	// Assert
	TestSuite.Test(__POUNAME()).AssertEqual(TEST_BOOL_TRUE, Success);
	TEST_DINT := 0;  // Buffer empty
	TestSuite.Test(__POUNAME()).AssertEqual(TEST_DINT, fbAnyBuffer.Metadata.elementCount);
END_IF
END_METHOD

// Element is removed but not copied when popDiscard=TRUE
METHOD PopDiscardTrue
VAR
	discardBuffer : BYTE;  // Can be any type when popDiscard=TRUE
END_VAR
IF TestSuite.Test(__POUNAME()).ExecuteTest() THEN
	// Arrange
	fbAnyBuffer.Clear();
	RawBuffer[TEST_LL+0] := 100;
	RawBuffer[TEST_LL+1] := 200;
	RawBuffer[TEST_LL+2] := 300;
	fbAnyBuffer.Metadata.elementCount := 3;
	discardBuffer := 0;

	// Act - Pop with discard=TRUE
	Success := fbAnyBuffer.PopRight(element := discardBuffer, popDiscard := TRUE);

	// Assert - Success but discardBuffer unchanged (no copy occurred)
	TestSuite.Test(__POUNAME()).AssertEqual(TEST_BOOL_TRUE, Success);
	TEST_DINT := 2;
	TestSuite.Test(__POUNAME()).AssertEqual(TEST_DINT, fbAnyBuffer.Metadata.elementCount);
	// Buffer should remain unchanged except last element cleared: [100, 200, 0]
	TEST_DINT := 100;
	TestSuite.Test(__POUNAME()).AssertEqual(TEST_DINT, RawBuffer[TEST_LL+0]);
	TEST_DINT := 200;
	TestSuite.Test(__POUNAME()).AssertEqual(TEST_DINT, RawBuffer[TEST_LL+1]);
	TEST_DINT := 0;
	TestSuite.Test(__POUNAME()).AssertEqual(TEST_DINT, RawBuffer[TEST_LL+2]);
END_IF
END_METHOD

// ElementCount decreases when popDiscard=TRUE
METHOD PopDiscardTrueDecrementsCount
VAR
	discardBuffer : DINT;
END_VAR
IF TestSuite.Test(__POUNAME()).ExecuteTest() THEN
	// Arrange
	fbAnyBuffer.Clear();
	RawBuffer[TEST_LL+0] := 100;
	RawBuffer[TEST_LL+1] := 200;
	RawBuffer[TEST_LL+2] := 300;
	fbAnyBuffer.Metadata.elementCount := 3;
	TEST_DINT := 3;
	TestSuite.Test(__POUNAME()).AssertEqual(TEST_DINT, fbAnyBuffer.Metadata.elementCount);

	// Act - Pop with discard=TRUE
	Success := fbAnyBuffer.PopRight(element := discardBuffer, popDiscard := TRUE);

	// Assert - Count decremented
	TestSuite.Test(__POUNAME()).AssertEqual(TEST_BOOL_TRUE, Success);
	TEST_DINT := 2;
	TestSuite.Test(__POUNAME()).AssertEqual(TEST_DINT, fbAnyBuffer.Metadata.elementCount);
END_IF
END_METHOD

// No element shifting occurs when popDiscard=TRUE (same as default)
METHOD PopDiscardTrueNoShift
VAR
	discardBuffer : DINT;
END_VAR
IF TestSuite.Test(__POUNAME()).ExecuteTest() THEN
	// Arrange
	fbAnyBuffer.Clear();
	RawBuffer[TEST_LL+0] := 10;
	RawBuffer[TEST_LL+1] := 20;
	RawBuffer[TEST_LL+2] := 30;
	RawBuffer[TEST_LL+3] := 40;
	fbAnyBuffer.Metadata.elementCount := 4;

	// Act - Pop with discard=TRUE
	Success := fbAnyBuffer.PopRight(element := discardBuffer, popDiscard := TRUE);

	// Assert - Elements stay in place (no shift)
	TestSuite.Test(__POUNAME()).AssertEqual(TEST_BOOL_TRUE, Success);
	TEST_DINT := 10;
	TestSuite.Test(__POUNAME()).AssertEqual(TEST_DINT, RawBuffer[TEST_LL+0]);
	TEST_DINT := 20;
	TestSuite.Test(__POUNAME()).AssertEqual(TEST_DINT, RawBuffer[TEST_LL+1]);
	TEST_DINT := 30;
	TestSuite.Test(__POUNAME()).AssertEqual(TEST_DINT, RawBuffer[TEST_LL+2]);
	TEST_DINT := 0;  // Last element cleared
	TestSuite.Test(__POUNAME()).AssertEqual(TEST_DINT, RawBuffer[TEST_LL+3]);
END_IF
END_METHOD

// No error when element size is wrong and popDiscard=TRUE
METHOD PopDiscardTrueSkipsTypeCheck
VAR
	wrongSizeBuffer : BYTE;  // Only 1 byte, but buffer expects DINT (4 bytes)
END_VAR
IF TestSuite.Test(__POUNAME()).ExecuteTest() THEN
	// Arrange
	fbAnyBuffer.Clear();
	RawBuffer[TEST_LL+0] := 100;
	RawBuffer[TEST_LL+1] := 200;
	fbAnyBuffer.Metadata.elementCount := 2;
	wrongSizeBuffer := 0;

	// Act - Pop with wrong type but popDiscard=TRUE (should succeed)
	Success := fbAnyBuffer.PopRight(element := wrongSizeBuffer, popDiscard := TRUE);

	// Assert - Should succeed despite type mismatch
	TestSuite.Test(__POUNAME()).AssertEqual(TEST_BOOL_TRUE, Success);
	TEST_DINT := 1;
	TestSuite.Test(__POUNAME()).AssertEqual(TEST_DINT, fbAnyBuffer.Metadata.elementCount);
END_IF
END_METHOD

// PopRight with wrong type succeeds when popDiscard=TRUE
METHOD PopDiscardWithWrongTypeSucceeds
VAR
	wrongTypeBuffer : INT;  // 2 bytes instead of 4
END_VAR
IF TestSuite.Test(__POUNAME()).ExecuteTest() THEN
	// Arrange
	fbAnyBuffer.Clear();
	RawBuffer[TEST_LL+0] := 999;
	RawBuffer[TEST_LL+1] := 888;
	fbAnyBuffer.Metadata.elementCount := 2;
	wrongTypeBuffer := 0;

	// Act - Pop with wrong type but popDiscard=TRUE
	Success := fbAnyBuffer.PopRight(element := wrongTypeBuffer, popDiscard := TRUE);

	// Assert - Should succeed
	TestSuite.Test(__POUNAME()).AssertEqual(TEST_BOOL_TRUE, Success);
	TEST_DINT := 1;
	TestSuite.Test(__POUNAME()).AssertEqual(TEST_DINT, fbAnyBuffer.Metadata.elementCount);
	// First element unchanged, last element cleared
	TEST_DINT := 999;
	TestSuite.Test(__POUNAME()).AssertEqual(TEST_DINT, RawBuffer[TEST_LL+0]);
	TEST_DINT := 0;
	TestSuite.Test(__POUNAME()).AssertEqual(TEST_DINT, RawBuffer[TEST_LL+1]);
END_IF
END_METHOD

// PopRight on empty buffer returns FALSE and does not modify buffer
METHOD PopFromEmptyBuffer
IF TestSuite.Test(__POUNAME()).ExecuteTest() THEN
	// Arrange - Clear buffer (elementCount = 0)
	fbAnyBuffer.Clear();
	ReturnedElement := 999;  // Set to non-zero to verify it is NOT overwritten

	// Act - Pop from empty buffer
	Success := fbAnyBuffer.PopRight(element := ReturnedElement);

	// Assert - Should fail because buffer is empty
	TestSuite.Test(__POUNAME()).AssertEqual(TEST_BOOL_FALSE, Success);

	// Element should remain unchanged (999) since pop failed
	TEST_DINT := 999;
	TestSuite.Test(__POUNAME()).AssertEqual(TEST_DINT, ReturnedElement);

	// All buffer positions should remain 0
	TEST_DINT := 0;
	TestSuite.Test(__POUNAME()).AssertEqual(TEST_DINT, RawBuffer[TEST_LL+0]);
	TestSuite.Test(__POUNAME()).AssertEqual(TEST_DINT, RawBuffer[TEST_LL+1]);
	TestSuite.Test(__POUNAME()).AssertEqual(TEST_DINT, RawBuffer[TEST_LL+2]);
	TestSuite.Test(__POUNAME()).AssertEqual(TEST_DINT, RawBuffer[TEST_LL+3]);
	TestSuite.Test(__POUNAME()).AssertEqual(TEST_DINT, RawBuffer[TEST_LL+4]);
END_IF
END_METHOD

// PopRight when buffer contains exactly one element
METHOD PopSingleElement
IF TestSuite.Test(__POUNAME()).ExecuteTest() THEN
	// Arrange - Only first element has data
	fbAnyBuffer.Clear();
	RawBuffer[TEST_LL+0] := 42;
	fbAnyBuffer.Metadata.elementCount := 1;
	ReturnedElement := 0;

	// Act
	Success := fbAnyBuffer.PopRight(element := ReturnedElement);

	// Assert - Should retrieve the single element
	TestSuite.Test(__POUNAME()).AssertEqual(TEST_BOOL_TRUE, Success);
	TEST_DINT := 42;
	TestSuite.Test(__POUNAME()).AssertEqual(TEST_DINT, ReturnedElement);

	// Buffer should now be completely empty
	TEST_DINT := 0;
	TestSuite.Test(__POUNAME()).AssertEqual(TEST_DINT, fbAnyBuffer.Metadata.elementCount);
	TestSuite.Test(__POUNAME()).AssertEqual(TEST_DINT, RawBuffer[TEST_LL+0]);
	TestSuite.Test(__POUNAME()).AssertEqual(TEST_DINT, RawBuffer[TEST_LL+1]);
	TestSuite.Test(__POUNAME()).AssertEqual(TEST_DINT, RawBuffer[TEST_LL+2]);
	TestSuite.Test(__POUNAME()).AssertEqual(TEST_DINT, RawBuffer[TEST_LL+3]);
	TestSuite.Test(__POUNAME()).AssertEqual(TEST_DINT, RawBuffer[TEST_LL+4]);
END_IF
END_METHOD

// PopRight can pop all elements until buffer is empty
METHOD PopUntilEmpty
VAR
	i : INT;
	ReturnedElement : DINT;
	testElement : DINT;
END_VAR
IF TestSuite.Test(__POUNAME()).ExecuteTest() THEN
	// Arrange - Fill buffer completely
	fbAnyBuffer.Clear();
	FOR i := 1 TO 5 DO
		testElement := TO_DINT(i * 100);
		fbAnyBuffer.PushRight(element := testElement);
	END_FOR

	// Act - Pop all elements
	FOR i := 5 TO 1 BY -1 DO
		Success := fbAnyBuffer.PopRight(element := ReturnedElement);
		TestSuite.Test(__POUNAME()).AssertEqual(TEST_BOOL_TRUE, Success);
		TEST_DINT := TO_DINT(i * 100);
		TestSuite.Test(__POUNAME()).AssertEqual(TEST_DINT, ReturnedElement);
	END_FOR

	// Assert - Buffer should be completely empty
	TEST_DINT := 0;
	TestSuite.Test(__POUNAME()).AssertEqual(TEST_DINT, fbAnyBuffer.Metadata.elementCount);

	// Try to pop from empty buffer
	Success := fbAnyBuffer.PopRight(element := ReturnedElement);
	TestSuite.Test(__POUNAME()).AssertEqual(TEST_BOOL_FALSE, Success);
END_IF
END_METHOD

// PopRight retrieves the last element from the buffer
METHOD RetrievesLastElement
IF TestSuite.Test(__POUNAME()).ExecuteTest() THEN
	// Arrange
	fbAnyBuffer.Clear();
	RawBuffer[TEST_LL+0] := 100;
	RawBuffer[TEST_LL+1] := 200;
	RawBuffer[TEST_LL+2] := 300;
	RawBuffer[TEST_LL+3] := 400;
	RawBuffer[TEST_LL+4] := 500;
	fbAnyBuffer.Metadata.elementCount := 5;
	ReturnedElement := 0;

	// Act
	Success := fbAnyBuffer.PopRight(element := ReturnedElement);

	// Assert
	TestSuite.Test(__POUNAME()).AssertEqual(TEST_BOOL_TRUE, Success);
	TEST_DINT := 500;
	TestSuite.Test(__POUNAME()).AssertEqual(TEST_DINT, ReturnedElement);
END_IF
END_METHOD

// PopRight returns TRUE when pop succeeds
METHOD ReturnsTrueOnSuccess
IF TestSuite.Test(__POUNAME()).ExecuteTest() THEN
	// Arrange
	fbAnyBuffer.Clear();
	RawBuffer[TEST_LL+0] := 100;
	fbAnyBuffer.Metadata.elementCount := 1;

	// Act
	Success := fbAnyBuffer.PopRight(element := ReturnedElement);

	// Assert
	TestSuite.Test(__POUNAME()).AssertEqual(TEST_BOOL_TRUE, Success);
END_IF
END_METHOD

// PopRight returns FALSE when element size doesn't match buffer element size
METHOD WrongSize
IF TestSuite.Test(__POUNAME()).ExecuteTest() THEN
	// Arrange
	fbAnyBuffer.Clear();
	RawBuffer[TEST_LL+0] := 100;
	fbAnyBuffer.Metadata.elementCount := 1;
	WrongSizeElement := 0;

	// Act - Pass an INT (2 bytes) to a DINT buffer (4 bytes)
	Success := fbAnyBuffer.PopRight(element := WrongSizeElement);

	// Assert
	TestSuite.Test(__POUNAME()).AssertEqual(TEST_BOOL_FALSE, Success);
END_IF
END_METHOD

END_PROGRAM

// ---- UnitTests/AnyBuffer/TEST_AnyBuffer_PushLeft.TcPOU
PROGRAM TEST_AnyBuffer_PushLeft

PushToEmptyBuffer();
PushToNonEmptyBuffer();
IncrementsElementCount();
ShiftsExistingElements();
ReturnsTrueOnSuccess();
ReturnsFalseOnFullBuffer();
ReturnsFalseOnWrongSize();
PreservesExistingData();
PushMultipleElements();
PushToFullBufferMinus1();
PushWhenFullCapacity();
PushZeroSizedElement();
PushWithDifferentDataTypes();
ConsecutivePushAndPopLeft();
ConsecutivePushAndPopRight();
ElementOrderAfterMultiplePushes();
FillBufferCompletely();

// LIFO behavior with alternating AppendLeft and PopLeft calls
METHOD ConsecutivePushAndPopLeft
VAR
	poppedValue : DINT;
END_VAR
IF TestSuite.Test(__POUNAME()).ExecuteTest() THEN
	// Arrange
	fbAnyBuffer.Clear();

	// Act - Append then Pop (LIFO: Last In First Out)
	AppendedElement := DINT#100;
	fbAnyBuffer.PushLeft(element := AppendedElement);  // [100]
	AppendedElement := DINT#200;
	fbAnyBuffer.PushLeft(element := AppendedElement);  // [200, 100]
	AppendedElement := DINT#300;
	fbAnyBuffer.PushLeft(element := AppendedElement);  // [300, 200, 100]
	fbAnyBuffer.PopLeft(element := poppedValue);  // Pop 300

	// Assert - Should pop the last appended value (300)
	TEST_DINT := 300;
	TestSuite.Test(__POUNAME()).AssertEqual(TEST_DINT, poppedValue);

	// Buffer should now be [200, 100]
	TEST_DINT := 200;
	TestSuite.Test(__POUNAME()).AssertEqual(TEST_DINT, RawBuffer[TEST_LL+0]);
	TEST_DINT := 100;
	TestSuite.Test(__POUNAME()).AssertEqual(TEST_DINT, RawBuffer[TEST_LL+1]);
	TEST_DINT := 2;
	TestSuite.Test(__POUNAME()).AssertEqual(TEST_DINT, fbAnyBuffer.Metadata.elementCount);
END_IF
END_METHOD

// FIFO behavior with alternating AppendLeft and PopRight calls
METHOD ConsecutivePushAndPopRight
VAR
	poppedValue : DINT;
END_VAR
IF TestSuite.Test(__POUNAME()).ExecuteTest() THEN
	// Arrange
	fbAnyBuffer.Clear();

	// Act - Append Left and Pop Right (FIFO from right)
	AppendedElement := DINT#100;
	fbAnyBuffer.PushLeft(element := AppendedElement);  // [100]
	AppendedElement := DINT#200;
	fbAnyBuffer.PushLeft(element := AppendedElement);  // [200, 100]
	AppendedElement := DINT#300;
	fbAnyBuffer.PushLeft(element := AppendedElement);  // [300, 200, 100]
	fbAnyBuffer.PopRight(element := poppedValue);  // Pop 100 (first appended)

	// Assert - Should pop the first appended value (100)
	TEST_DINT := 100;
	TestSuite.Test(__POUNAME()).AssertEqual(TEST_DINT, poppedValue);

	// Buffer should now be [300, 200]
	TEST_DINT := 300;
	TestSuite.Test(__POUNAME()).AssertEqual(TEST_DINT, RawBuffer[TEST_LL+0]);
	TEST_DINT := 200;
	TestSuite.Test(__POUNAME()).AssertEqual(TEST_DINT, RawBuffer[TEST_LL+1]);
	TEST_DINT := 2;
	TestSuite.Test(__POUNAME()).AssertEqual(TEST_DINT, fbAnyBuffer.Metadata.elementCount);
END_IF
END_METHOD

// AppendLeft maintains correct element order after multiple appends
METHOD ElementOrderAfterMultiplePushes
IF TestSuite.Test(__POUNAME()).ExecuteTest() THEN
	// Arrange
	fbAnyBuffer.Clear();

	// Act - Append 5 different values
	AppendedElement := DINT#1;
	fbAnyBuffer.PushLeft(element := AppendedElement);    // [1]
	AppendedElement := DINT#2;
	fbAnyBuffer.PushLeft(element := AppendedElement);    // [2, 1]
	AppendedElement := DINT#3;
	fbAnyBuffer.PushLeft(element := AppendedElement);    // [3, 2, 1]
	AppendedElement := DINT#4;
	fbAnyBuffer.PushLeft(element := AppendedElement);    // [4, 3, 2, 1]
	AppendedElement := DINT#5;
	fbAnyBuffer.PushLeft(element := AppendedElement);    // [5, 4, 3, 2, 1]

	// Assert - Verify complete LIFO order
	TEST_DINT := 5;
	TestSuite.Test(__POUNAME()).AssertEqual(TEST_DINT, RawBuffer[TEST_LL+0]);
	TEST_DINT := 4;
	TestSuite.Test(__POUNAME()).AssertEqual(TEST_DINT, RawBuffer[TEST_LL+1]);
	TEST_DINT := 3;
	TestSuite.Test(__POUNAME()).AssertEqual(TEST_DINT, RawBuffer[TEST_LL+2]);
	TEST_DINT := 2;
	TestSuite.Test(__POUNAME()).AssertEqual(TEST_DINT, RawBuffer[TEST_LL+3]);
	TEST_DINT := 1;
	TestSuite.Test(__POUNAME()).AssertEqual(TEST_DINT, RawBuffer[TEST_LL+4]);
	TEST_DINT := 5;
	TestSuite.Test(__POUNAME()).AssertEqual(TEST_DINT, fbAnyBuffer.Metadata.elementCount);
END_IF
END_METHOD

// Filling buffer to full capacity works correctly
METHOD FillBufferCompletely
VAR
	i : INT;
END_VAR
IF TestSuite.Test(__POUNAME()).ExecuteTest() THEN
	// Arrange
	fbAnyBuffer.Clear();

	// Act - Fill buffer completely
	FOR i := 1 TO 5 DO
		AppendedElement := TO_DINT(i * 100);
		Success := fbAnyBuffer.PushLeft(element := AppendedElement);
		TestSuite.Test(__POUNAME()).AssertEqual(TEST_BOOL_TRUE, Success);
	END_FOR

	// Assert - All elements in correct positions (reverse order due to left append)
	TEST_DINT := 500;
	TestSuite.Test(__POUNAME()).AssertEqual(TEST_DINT, RawBuffer[TEST_LL+0]);
	TEST_DINT := 400;
	TestSuite.Test(__POUNAME()).AssertEqual(TEST_DINT, RawBuffer[TEST_LL+1]);
	TEST_DINT := 300;
	TestSuite.Test(__POUNAME()).AssertEqual(TEST_DINT, RawBuffer[TEST_LL+2]);
	TEST_DINT := 200;
	TestSuite.Test(__POUNAME()).AssertEqual(TEST_DINT, RawBuffer[TEST_LL+3]);
	TEST_DINT := 100;
	TestSuite.Test(__POUNAME()).AssertEqual(TEST_DINT, RawBuffer[TEST_LL+4]);
	TEST_DINT := 5;
	TestSuite.Test(__POUNAME()).AssertEqual(TEST_DINT, fbAnyBuffer.Metadata.elementCount);

	// Assert - Cannot append when full
	AppendedElement := DINT#600;
	Success := fbAnyBuffer.PushLeft(element := AppendedElement);
	TestSuite.Test(__POUNAME()).AssertEqual(TEST_BOOL_FALSE, Success);
END_IF
END_METHOD

// AppendLeft increases elementCount by 1 after append
METHOD IncrementsElementCount
IF TestSuite.Test(__POUNAME()).ExecuteTest() THEN
	// Arrange
	fbAnyBuffer.Clear();
	RawBuffer[TEST_LL+0] := 100;
	RawBuffer[TEST_LL+1] := 200;
	fbAnyBuffer.Metadata.elementCount := 2;
	AppendedElement := 300;

	// Act
	Success := fbAnyBuffer.PushLeft(element := AppendedElement);

	// Assert - elementCount should be incremented from 2 to 3
	TEST_DINT := 3;
	TestSuite.Test(__POUNAME()).AssertEqual(TEST_DINT, fbAnyBuffer.Metadata.elementCount);
END_IF
END_METHOD

// AppendLeft preserves existing element values after shift
METHOD PreservesExistingData
IF TestSuite.Test(__POUNAME()).ExecuteTest() THEN
	// Arrange
	fbAnyBuffer.Clear();
	RawBuffer[TEST_LL+0] := 111;
	RawBuffer[TEST_LL+1] := 222;
	RawBuffer[TEST_LL+2] := 333;
	fbAnyBuffer.Metadata.elementCount := 3;
	AppendedElement := 999;

	// Act
	Success := fbAnyBuffer.PushLeft(element := AppendedElement);

	// Assert - All original values preserved (just shifted)
	TEST_DINT := 999;
	TestSuite.Test(__POUNAME()).AssertEqual(TEST_DINT, RawBuffer[TEST_LL+0]);
	TEST_DINT := 111;
	TestSuite.Test(__POUNAME()).AssertEqual(TEST_DINT, RawBuffer[TEST_LL+1]);
	TEST_DINT := 222;
	TestSuite.Test(__POUNAME()).AssertEqual(TEST_DINT, RawBuffer[TEST_LL+2]);
	TEST_DINT := 333;
	TestSuite.Test(__POUNAME()).AssertEqual(TEST_DINT, RawBuffer[TEST_LL+3]);
END_IF
END_METHOD

// AppendLeft consecutive appends work correctly (LIFO order)
METHOD PushMultipleElements
IF TestSuite.Test(__POUNAME()).ExecuteTest() THEN
	// Arrange
	fbAnyBuffer.Clear();

	// Act - Append multiple elements to the left (stack behavior)
	AppendedElement := DINT#10;
	fbAnyBuffer.PushLeft(element := AppendedElement);
	AppendedElement := DINT#20;
	fbAnyBuffer.PushLeft(element := AppendedElement);
	AppendedElement := DINT#30;
	fbAnyBuffer.PushLeft(element := AppendedElement);

	// Assert - LIFO order: last appended (30) should be at position 0
	TEST_DINT := 30;
	TestSuite.Test(__POUNAME()).AssertEqual(TEST_DINT, RawBuffer[TEST_LL+0]);
	TEST_DINT := 20;
	TestSuite.Test(__POUNAME()).AssertEqual(TEST_DINT, RawBuffer[TEST_LL+1]);
	TEST_DINT := 10;
	TestSuite.Test(__POUNAME()).AssertEqual(TEST_DINT, RawBuffer[TEST_LL+2]);
	TEST_DINT := 3;
	TestSuite.Test(__POUNAME()).AssertEqual(TEST_DINT, fbAnyBuffer.Metadata.elementCount);
END_IF
END_METHOD

// AppendLeft inserts element at position 0 in empty buffer
METHOD PushToEmptyBuffer
IF TestSuite.Test(__POUNAME()).ExecuteTest() THEN
	// Arrange
	fbAnyBuffer.Clear();
	AppendedElement := 100;

	// Act
	Success := fbAnyBuffer.PushLeft(element := AppendedElement);

	// Assert
	TestSuite.Test(__POUNAME()).AssertEqual(TEST_BOOL_TRUE, Success);
	TEST_DINT := 100;
	TestSuite.Test(__POUNAME()).AssertEqual(TEST_DINT, RawBuffer[TEST_LL+0]);
	TEST_DINT := 1;
	TestSuite.Test(__POUNAME()).AssertEqual(TEST_DINT, fbAnyBuffer.Metadata.elementCount);
END_IF
END_METHOD

// AppendLeft succeeds when buffer has exactly 1 space remaining
METHOD PushToFullBufferMinus1
IF TestSuite.Test(__POUNAME()).ExecuteTest() THEN
	// Arrange - Fill buffer with 4 elements (capacity is 5)
	fbAnyBuffer.Clear();
	RawBuffer[TEST_LL+0] := 100;
	RawBuffer[TEST_LL+1] := 200;
	RawBuffer[TEST_LL+2] := 300;
	RawBuffer[TEST_LL+3] := 400;
	fbAnyBuffer.Metadata.elementCount := 4;
	AppendedElement := 50;

	// Act - Append to buffer with exactly 1 space left
	Success := fbAnyBuffer.PushLeft(element := AppendedElement);

	// Assert
	TestSuite.Test(__POUNAME()).AssertEqual(TEST_BOOL_TRUE, Success);
	TEST_DINT := 5;
	TestSuite.Test(__POUNAME()).AssertEqual(TEST_DINT, fbAnyBuffer.Metadata.elementCount);
	TEST_DINT := 50;
	TestSuite.Test(__POUNAME()).AssertEqual(TEST_DINT, RawBuffer[TEST_LL+0]);
END_IF
END_METHOD

// AppendLeft inserts element at position 0 and shifts existing elements right
METHOD PushToNonEmptyBuffer
IF TestSuite.Test(__POUNAME()).ExecuteTest() THEN
	// Arrange
	fbAnyBuffer.Clear();
	RawBuffer[TEST_LL+0] := 200;
	RawBuffer[TEST_LL+1] := 300;
	fbAnyBuffer.Metadata.capacity := 3;
	fbAnyBuffer.Metadata.elementCount := 2;
	AppendedElement := 100;

	// Act
	Success := fbAnyBuffer.PushLeft(element := AppendedElement);

	// Assert
	TestSuite.Test(__POUNAME()).AssertEqual(TEST_BOOL_TRUE, Success);
	TEST_DINT := 100;
	TestSuite.Test(__POUNAME()).AssertEqual(TEST_DINT, RawBuffer[TEST_LL+0]);
	TEST_DINT := 200;
	TestSuite.Test(__POUNAME()).AssertEqual(TEST_DINT, RawBuffer[TEST_LL+1]);
	TEST_DINT := 300;
	TestSuite.Test(__POUNAME()).AssertEqual(TEST_DINT, RawBuffer[TEST_LL+2]);
END_IF
END_METHOD

// AppendLeft fails when elementCount equals capacity
METHOD PushWhenFullCapacity
IF TestSuite.Test(__POUNAME()).ExecuteTest() THEN
	// Arrange - Set elementCount to capacity
	// Arrange - Fill buffer to capacity (5 elements)
	fbAnyBuffer.Clear();
	RawBuffer[TEST_LL+0] := 100;
	RawBuffer[TEST_LL+1] := 200;
	RawBuffer[TEST_LL+2] := 300;
	RawBuffer[TEST_LL+3] := 400;
	RawBuffer[TEST_LL+4] := 500;
	fbAnyBuffer.Metadata.elementCount := TEST_UL-TEST_LL+1;
	fbAnyBuffer.Metadata.capacity := 0;
	AppendedElement := 999;

	// Act
	Success := fbAnyBuffer.PushLeft(element := AppendedElement);

	// Assert
	TestSuite.Test(__POUNAME()).AssertEqual(TEST_BOOL_FALSE, Success);
	TEST_DINT := 5;
	TestSuite.Test(__POUNAME()).AssertEqual(TEST_DINT, fbAnyBuffer.Metadata.elementCount);
END_IF
END_METHOD

// AppendLeft works with various data types (DINT, REAL, struct)
METHOD PushWithDifferentDataTypes
VAR
	realBuffer : ARRAY[0..4] OF REAL;
	fbRealBuffer : AnyBuffer(pBuffer := realBuffer,
								bufferBoundLower := 0,
								bufferBoundUpper := 4,
								isBufferPersistent := FALSE);
	realValue : REAL := 3.14159;
	retrievedReal : REAL;
END_VAR
IF TestSuite.Test(__POUNAME()).ExecuteTest() THEN
	// Arrange
	fbRealBuffer.Clear();
	realValue := 3.14159;

	// Act - Append REAL type
	Success := fbRealBuffer.PushLeft(element := realValue);

	// Assert
	TestSuite.Test(__POUNAME()).AssertEqual(TEST_BOOL_TRUE, Success);
	TEST_REAL := 3.14159;
	TestSuite.Test(__POUNAME()).AssertEqual(TEST_REAL, realBuffer[0]);
END_IF
END_METHOD

// AppendLeft with zero-sized element
METHOD PushZeroSizedElement
VAR
	EmptyAny				: __SYSTEM.AnyType;
END_VAR
IF TestSuite.Test(__POUNAME()).ExecuteTest() THEN
	// Arrange
	fbAnyBuffer.Clear();

	// Initialize empty AnyType (size = 0)
	EmptyAny.pValue := 0;
	EmptyAny.diSize := 0;

	// Act - Call with zero-sized element
	Success := fbAnyBuffer.PushLeft(element := EmptyAny);

	// Assert - Should fail because element size doesn't match
	TestSuite.Test(__POUNAME()).AssertEqual(TEST_BOOL_FALSE, Success);
END_IF
END_METHOD

// AppendLeft returns FALSE when buffer is at capacity
METHOD ReturnsFalseOnFullBuffer
IF TestSuite.Test(__POUNAME()).ExecuteTest() THEN
	// Arrange - Fill buffer to capacity (5 elements)
	fbAnyBuffer.Clear();
	RawBuffer[TEST_LL+0] := 100;
	RawBuffer[TEST_LL+1] := 200;
	RawBuffer[TEST_LL+2] := 300;
	RawBuffer[TEST_LL+3] := 400;
	RawBuffer[TEST_LL+4] := 500;
	fbAnyBuffer.Metadata.elementCount := TEST_UL+1;
	fbAnyBuffer.Metadata.capacity := 0;
	AppendedElement := 600;

	// Act - Try to append to full buffer
	Success := fbAnyBuffer.PushLeft(element := AppendedElement);

	// Assert
	TestSuite.Test(__POUNAME()).AssertEqual(TEST_BOOL_FALSE, Success);
	// Verify buffer unchanged
	TEST_DINT := 100;
	TestSuite.Test(__POUNAME()).AssertEqual(TEST_DINT, RawBuffer[TEST_LL+0]);
END_IF
END_METHOD

// AppendLeft returns FALSE when element size doesn't match buffer element size
METHOD ReturnsFalseOnWrongSize
IF TestSuite.Test(__POUNAME()).ExecuteTest() THEN
	// Arrange
	fbAnyBuffer.Clear();
	WrongSizeElement := 100;  // INT is 2 bytes, buffer expects DINT (4 bytes)

	// Act - Pass an INT to a DINT buffer
	Success := fbAnyBuffer.PushLeft(element := WrongSizeElement);

	// Assert
	TestSuite.Test(__POUNAME()).AssertEqual(TEST_BOOL_FALSE, Success);
END_IF
END_METHOD

// AppendLeft returns TRUE when append succeeds
METHOD ReturnsTrueOnSuccess
IF TestSuite.Test(__POUNAME()).ExecuteTest() THEN
	// Arrange
	fbAnyBuffer.Clear();
	AppendedElement := 42;

	// Act
	Success := fbAnyBuffer.PushLeft(element := AppendedElement);

	// Assert
	TestSuite.Test(__POUNAME()).AssertEqual(TEST_BOOL_TRUE, Success);
END_IF
END_METHOD

// AppendLeft shifts all existing elements right by one position
METHOD ShiftsExistingElements
IF TestSuite.Test(__POUNAME()).ExecuteTest() THEN
	// Arrange
	fbAnyBuffer.Clear();
	RawBuffer[TEST_LL+0] := 100;
	RawBuffer[TEST_LL+1] := 200;
	RawBuffer[TEST_LL+2] := 300;
	fbAnyBuffer.Metadata.elementCount := 3;
	AppendedElement := 50;

	// Act
	Success := fbAnyBuffer.PushLeft(element := AppendedElement);

	// Assert - all elements shifted right
	TEST_DINT := 50;
	TestSuite.Test(__POUNAME()).AssertEqual(TEST_DINT, RawBuffer[TEST_LL+0]);
	TEST_DINT := 100;
	TestSuite.Test(__POUNAME()).AssertEqual(TEST_DINT, RawBuffer[TEST_LL+1]);
	TEST_DINT := 200;
	TestSuite.Test(__POUNAME()).AssertEqual(TEST_DINT, RawBuffer[TEST_LL+2]);
	TEST_DINT := 300;
	TestSuite.Test(__POUNAME()).AssertEqual(TEST_DINT, RawBuffer[TEST_LL+3]);
END_IF
END_METHOD

END_PROGRAM

// ---- UnitTests/AnyBuffer/TEST_AnyBuffer_PushRight.TcPOU
PROGRAM TEST_AnyBuffer_PushRight

PushToEmptyBuffer();
PushToNonEmptyBuffer();
IncrementsElementCount();
DoesNotShiftElements();
ReturnsTrueOnSuccess();
ReturnsFalseOnFullBuffer();
ReturnsFalseOnWrongSize();
PreservesExistingData();
PushMultipleElements();
PushToFullBufferMinus1();
PushWhenFullCapacity();
PushZeroSizedElement();
PushWithDifferentDataTypes();
ConsecutivePushAndPopLeft();
ConsecutivePushAndPopRight();
ElementOrderAfterMultiplePushes();
FillBufferCompletely();

// AppendRight and PopLeft demonstrate FIFO behavior
METHOD ConsecutivePushAndPopLeft
VAR
	ReturnedElement : DINT;
END_VAR
IF TestSuite.Test(__POUNAME()).ExecuteTest() THEN
	// Arrange
	fbAnyBuffer.Clear();

	// Act - Append then Pop (FIFO: First In First Out)
	testElement := DINT#100;
	fbAnyBuffer.PushRight(element := testElement);  // [100]
	testElement := DINT#200;
	fbAnyBuffer.PushRight(element := testElement);  // [100, 200]
	testElement := DINT#300;
	fbAnyBuffer.PushRight(element := testElement);  // [100, 200, 300]
	fbAnyBuffer.PopLeft(element := ReturnedElement);   // Pop 100

	// Assert - Should pop the first appended value (100)
	TEST_DINT := 100;
	TestSuite.Test(__POUNAME()).AssertEqual(TEST_DINT, ReturnedElement);

	// Buffer should now be [200, 300]
	TEST_DINT := 200;
	TestSuite.Test(__POUNAME()).AssertEqual(TEST_DINT, RawBuffer[TEST_LL+0]);
	TEST_DINT := 300;
	TestSuite.Test(__POUNAME()).AssertEqual(TEST_DINT, RawBuffer[TEST_LL+1]);
END_IF
END_METHOD

// AppendRight and PopRight demonstrate LIFO behavior
METHOD ConsecutivePushAndPopRight
VAR
	ReturnedElement : DINT;
END_VAR
IF TestSuite.Test(__POUNAME()).ExecuteTest() THEN
	// Arrange
	fbAnyBuffer.Clear();

	// Act - Append then Pop from right (LIFO: Last In First Out)
	testElement := DINT#100;
	fbAnyBuffer.PushRight(element := testElement);  // [100]
	testElement := DINT#200;
	fbAnyBuffer.PushRight(element := testElement);  // [100, 200]
	testElement := DINT#300;
	fbAnyBuffer.PushRight(element := testElement);  // [100, 200, 300]
	fbAnyBuffer.PopRight(element := ReturnedElement);  // Pop 300

	// Assert - Should pop the last appended value (300)
	TEST_DINT := 300;
	TestSuite.Test(__POUNAME()).AssertEqual(TEST_DINT, ReturnedElement);

	// Buffer should now be [100, 200]
	TEST_DINT := 100;
	TestSuite.Test(__POUNAME()).AssertEqual(TEST_DINT, RawBuffer[TEST_LL+0]);
	TEST_DINT := 200;
	TestSuite.Test(__POUNAME()).AssertEqual(TEST_DINT, RawBuffer[TEST_LL+1]);
END_IF
END_METHOD

// AppendRight does not move any existing elements
METHOD DoesNotShiftElements
IF TestSuite.Test(__POUNAME()).ExecuteTest() THEN
	// Arrange
	fbAnyBuffer.Clear();
	RawBuffer[TEST_LL+0] := 111;
	RawBuffer[TEST_LL+1] := 222;
	RawBuffer[TEST_LL+2] := 333;
	fbAnyBuffer.Metadata.elementCount := 3;
	AppendedElement := 444;

	// Act
	Success := fbAnyBuffer.PushRight(element := AppendedElement);

	// Assert - all existing elements remain at their original positions
	TEST_DINT := 111;
	TestSuite.Test(__POUNAME()).AssertEqual(TEST_DINT, RawBuffer[TEST_LL+0]);
	TEST_DINT := 222;
	TestSuite.Test(__POUNAME()).AssertEqual(TEST_DINT, RawBuffer[TEST_LL+1]);
	TEST_DINT := 333;
	TestSuite.Test(__POUNAME()).AssertEqual(TEST_DINT, RawBuffer[TEST_LL+2]);
	TEST_DINT := 444;
	TestSuite.Test(__POUNAME()).AssertEqual(TEST_DINT, RawBuffer[TEST_LL+3]);
END_IF
END_METHOD

// AppendRight maintains correct element order after multiple appends
METHOD ElementOrderAfterMultiplePushes
IF TestSuite.Test(__POUNAME()).ExecuteTest() THEN
	// Arrange
	fbAnyBuffer.Clear();

	// Act - Append 5 different values
	testElement := DINT#1;
	fbAnyBuffer.PushRight(element := testElement);    // [1]
	testElement := DINT#2;
	fbAnyBuffer.PushRight(element := testElement);    // [1, 2]
	testElement := DINT#3;
	fbAnyBuffer.PushRight(element := testElement);    // [1, 2, 3]
	testElement := DINT#4;
	fbAnyBuffer.PushRight(element := testElement);    // [1, 2, 3, 4]
	testElement := DINT#5;
	fbAnyBuffer.PushRight(element := testElement);    // [1, 2, 3, 4, 5]

	// Assert - Verify sequential order
	TEST_DINT := 1;
	TestSuite.Test(__POUNAME()).AssertEqual(TEST_DINT, RawBuffer[TEST_LL+0]);
	TEST_DINT := 2;
	TestSuite.Test(__POUNAME()).AssertEqual(TEST_DINT, RawBuffer[TEST_LL+1]);
	TEST_DINT := 3;
	TestSuite.Test(__POUNAME()).AssertEqual(TEST_DINT, RawBuffer[TEST_LL+2]);
	TEST_DINT := 4;
	TestSuite.Test(__POUNAME()).AssertEqual(TEST_DINT, RawBuffer[TEST_LL+3]);
	TEST_DINT := 5;
	TestSuite.Test(__POUNAME()).AssertEqual(TEST_DINT, RawBuffer[TEST_LL+4]);
	TEST_DINT := 5;
	TestSuite.Test(__POUNAME()).AssertEqual(TEST_DINT, fbAnyBuffer.Metadata.elementCount);
END_IF
END_METHOD

// AppendRight can fill buffer to full capacity correctly
METHOD FillBufferCompletely
VAR
	i : INT;
END_VAR
IF TestSuite.Test(__POUNAME()).ExecuteTest() THEN
	// Arrange
	fbAnyBuffer.Clear();

	// Act - Fill buffer completely
	FOR i := 1 TO 5 DO
		testElement := TO_DINT(i * 100);
		Success := fbAnyBuffer.PushRight(element := testElement);
		TestSuite.Test(__POUNAME()).AssertEqual(TEST_BOOL_TRUE, Success);
	END_FOR

	// Assert - All elements in correct positions
	TEST_DINT := 100;
	TestSuite.Test(__POUNAME()).AssertEqual(TEST_DINT, RawBuffer[TEST_LL+0]);
	TEST_DINT := 200;
	TestSuite.Test(__POUNAME()).AssertEqual(TEST_DINT, RawBuffer[TEST_LL+1]);
	TEST_DINT := 300;
	TestSuite.Test(__POUNAME()).AssertEqual(TEST_DINT, RawBuffer[TEST_LL+2]);
	TEST_DINT := 400;
	TestSuite.Test(__POUNAME()).AssertEqual(TEST_DINT, RawBuffer[TEST_LL+3]);
	TEST_DINT := 500;
	TestSuite.Test(__POUNAME()).AssertEqual(TEST_DINT, RawBuffer[TEST_LL+4]);
	TEST_DINT := 5;
	TestSuite.Test(__POUNAME()).AssertEqual(TEST_DINT, fbAnyBuffer.Metadata.elementCount);

	// Assert - Cannot append when full
	testElement := DINT#600;
	Success := fbAnyBuffer.PushRight(element := testElement);
	TestSuite.Test(__POUNAME()).AssertEqual(TEST_BOOL_FALSE, Success);
END_IF
END_METHOD

// AppendRight increases elementCount by 1 after append
METHOD IncrementsElementCount
IF TestSuite.Test(__POUNAME()).ExecuteTest() THEN
	// Arrange
	fbAnyBuffer.Clear();
	RawBuffer[TEST_LL+0] := 100;
	RawBuffer[TEST_LL+1] := 200;
	fbAnyBuffer.Metadata.elementCount := 2;
	AppendedElement := 300;

	// Act
	Success := fbAnyBuffer.PushRight(element := AppendedElement);

	// Assert - elementCount should be incremented from 2 to 3
	TEST_DINT := 3;
	TestSuite.Test(__POUNAME()).AssertEqual(TEST_DINT, fbAnyBuffer.Metadata.elementCount);
END_IF
END_METHOD

// AppendRight preserves existing element values
METHOD PreservesExistingData
IF TestSuite.Test(__POUNAME()).ExecuteTest() THEN
	// Arrange
	fbAnyBuffer.Clear();
	RawBuffer[TEST_LL+0] := 111;
	RawBuffer[TEST_LL+1] := 222;
	RawBuffer[TEST_LL+2] := 333;
	fbAnyBuffer.Metadata.elementCount := 3;
	AppendedElement := 999;

	// Act
	Success := fbAnyBuffer.PushRight(element := AppendedElement);

	// Assert - All original values preserved (not shifted)
	TEST_DINT := 111;
	TestSuite.Test(__POUNAME()).AssertEqual(TEST_DINT, RawBuffer[TEST_LL+0]);
	TEST_DINT := 222;
	TestSuite.Test(__POUNAME()).AssertEqual(TEST_DINT, RawBuffer[TEST_LL+1]);
	TEST_DINT := 333;
	TestSuite.Test(__POUNAME()).AssertEqual(TEST_DINT, RawBuffer[TEST_LL+2]);
	TEST_DINT := 999;
	TestSuite.Test(__POUNAME()).AssertEqual(TEST_DINT, RawBuffer[TEST_LL+3]);
END_IF
END_METHOD

// AppendRight consecutive appends work correctly (FIFO order with PopLeft)
METHOD PushMultipleElements
IF TestSuite.Test(__POUNAME()).ExecuteTest() THEN
	// Arrange
	fbAnyBuffer.Clear();

	// Act - Append multiple elements to the right (queue behavior)
	testElement := DINT#10;
	fbAnyBuffer.PushRight(element := testElement);
	testElement := DINT#20;
	fbAnyBuffer.PushRight(element := testElement);
	testElement := DINT#30;
	fbAnyBuffer.PushRight(element := testElement);

	// Assert - Sequential order: elements appear in order appended
	TEST_DINT := 10;
	TestSuite.Test(__POUNAME()).AssertEqual(TEST_DINT, RawBuffer[TEST_LL+0]);
	TEST_DINT := 20;
	TestSuite.Test(__POUNAME()).AssertEqual(TEST_DINT, RawBuffer[TEST_LL+1]);
	TEST_DINT := 30;
	TestSuite.Test(__POUNAME()).AssertEqual(TEST_DINT, RawBuffer[TEST_LL+2]);
	TEST_DINT := 3;
	TestSuite.Test(__POUNAME()).AssertEqual(TEST_DINT, fbAnyBuffer.Metadata.elementCount);
END_IF
END_METHOD

// AppendRight inserts element at position 0 in empty buffer
METHOD PushToEmptyBuffer
IF TestSuite.Test(__POUNAME()).ExecuteTest() THEN
	// Arrange
	fbAnyBuffer.Clear();
	AppendedElement := 100;

	// Act
	Success := fbAnyBuffer.PushRight(element := AppendedElement);

	// Assert
	TestSuite.Test(__POUNAME()).AssertEqual(TEST_BOOL_TRUE, Success);
	TEST_DINT := 100;
	TestSuite.Test(__POUNAME()).AssertEqual(TEST_DINT, RawBuffer[TEST_LL+0]);
	TEST_DINT := 1;
	TestSuite.Test(__POUNAME()).AssertEqual(TEST_DINT, fbAnyBuffer.Metadata.elementCount);
END_IF
END_METHOD

// AppendRight succeeds when buffer has exactly 1 space remaining
METHOD PushToFullBufferMinus1
IF TestSuite.Test(__POUNAME()).ExecuteTest() THEN
	// Arrange - Fill buffer with 4 elements (capacity is 5)
	fbAnyBuffer.Clear();
	RawBuffer[TEST_LL+0] := 100;
	RawBuffer[TEST_LL+1] := 200;
	RawBuffer[TEST_LL+2] := 300;
	RawBuffer[TEST_LL+3] := 400;
	fbAnyBuffer.Metadata.elementCount := 4;
	AppendedElement := 500;

	// Act - Append to buffer with exactly 1 space left
	Success := fbAnyBuffer.PushRight(element := AppendedElement);

	// Assert
	TestSuite.Test(__POUNAME()).AssertEqual(TEST_BOOL_TRUE, Success);
	TEST_DINT := 5;
	TestSuite.Test(__POUNAME()).AssertEqual(TEST_DINT, fbAnyBuffer.Metadata.elementCount);
	TEST_DINT := 500;
	TestSuite.Test(__POUNAME()).AssertEqual(TEST_DINT, RawBuffer[TEST_LL+4]);
END_IF
END_METHOD

// AppendRight inserts element at position elementCount and no elements shift
METHOD PushToNonEmptyBuffer
IF TestSuite.Test(__POUNAME()).ExecuteTest() THEN
	// Arrange
	fbAnyBuffer.Clear();
	RawBuffer[TEST_LL+0] := 100;
	RawBuffer[TEST_LL+1] := 200;
	fbAnyBuffer.Metadata.capacity := 3;
	fbAnyBuffer.Metadata.elementCount := 2;
	AppendedElement := 300;

	// Act
	Success := fbAnyBuffer.PushRight(element := AppendedElement);

	// Assert
	TestSuite.Test(__POUNAME()).AssertEqual(TEST_BOOL_TRUE, Success);
	TEST_DINT := 100;
	TestSuite.Test(__POUNAME()).AssertEqual(TEST_DINT, RawBuffer[TEST_LL+0]);
	TEST_DINT := 200;
	TestSuite.Test(__POUNAME()).AssertEqual(TEST_DINT, RawBuffer[TEST_LL+1]);
	TEST_DINT := 300;
	TestSuite.Test(__POUNAME()).AssertEqual(TEST_DINT, RawBuffer[TEST_LL+2]);
END_IF
END_METHOD

// AppendRight fails when elementCount equals capacity
METHOD PushWhenFullCapacity
IF TestSuite.Test(__POUNAME()).ExecuteTest() THEN
	// Arrange - Fill buffer to capacity (5 elements)
	fbAnyBuffer.Clear();
	RawBuffer[TEST_LL+0] := 100;
	RawBuffer[TEST_LL+1] := 200;
	RawBuffer[TEST_LL+2] := 300;
	RawBuffer[TEST_LL+3] := 400;
	RawBuffer[TEST_LL+4] := 500;
	fbAnyBuffer.Metadata.elementCount := TEST_UL-TEST_LL+1;
	fbAnyBuffer.Metadata.capacity := 0;
	AppendedElement := 999;

	// Act
	Success := fbAnyBuffer.PushRight(element := AppendedElement);

	// Assert
	TestSuite.Test(__POUNAME()).AssertEqual(TEST_BOOL_FALSE, Success);
	TEST_DINT := 5;
	TestSuite.Test(__POUNAME()).AssertEqual(TEST_DINT, fbAnyBuffer.Metadata.elementCount);
END_IF
END_METHOD

// AppendRight works with various data types (DINT, REAL, struct)
METHOD PushWithDifferentDataTypes
VAR
	realBuffer : ARRAY[0..4] OF REAL;
	fbRealBuffer : AnyBuffer(pBuffer := realBuffer,
								bufferBoundLower := 0,
								bufferBoundUpper := 4,
								isBufferPersistent := FALSE);
	realValue : REAL := 3.14159;
	retrievedReal : REAL;
END_VAR
IF TestSuite.Test(__POUNAME()).ExecuteTest() THEN
	// Arrange
	fbRealBuffer.Clear();
	realValue := 3.14159;

	// Act - Append REAL type
	Success := fbRealBuffer.PushRight(element := realValue);

	// Assert
	TestSuite.Test(__POUNAME()).AssertEqual(TEST_BOOL_TRUE, Success);
	TEST_REAL := 3.14159;
	TestSuite.Test(__POUNAME()).AssertEqual(TEST_REAL, realBuffer[0]);
END_IF
END_METHOD

// AppendRight with zero-sized element
METHOD PushZeroSizedElement
VAR
	EmptyAny				: __SYSTEM.AnyType;
END_VAR
IF TestSuite.Test(__POUNAME()).ExecuteTest() THEN
	// Arrange
	fbAnyBuffer.Clear();

	// Initialize empty AnyType (size = 0)
	EmptyAny.pValue := 0;
	EmptyAny.diSize := 0;

	// Act - Call with zero-sized element
	Success := fbAnyBuffer.PushRight(element := EmptyAny);

	// Assert - Should fail because element size doesn't match
	TestSuite.Test(__POUNAME()).AssertEqual(TEST_BOOL_FALSE, Success);
END_IF
END_METHOD

// AppendRight returns FALSE when buffer is at capacity
METHOD ReturnsFalseOnFullBuffer
IF TestSuite.Test(__POUNAME()).ExecuteTest() THEN
	// Arrange - Fill buffer to capacity (5 elements)
	fbAnyBuffer.Clear();
	RawBuffer[TEST_LL+0] := 100;
	RawBuffer[TEST_LL+1] := 200;
	RawBuffer[TEST_LL+2] := 300;
	RawBuffer[TEST_LL+3] := 400;
	RawBuffer[TEST_LL+4] := 500;
	fbAnyBuffer.Metadata.elementCount := TEST_UL+1;
	fbAnyBuffer.Metadata.capacity := 0;
	AppendedElement := 600;

	// Act - Try to append to full buffer
	Success := fbAnyBuffer.PushRight(element := AppendedElement);

	// Assert
	TestSuite.Test(__POUNAME()).AssertEqual(TEST_BOOL_FALSE, Success);
	// Verify buffer unchanged
	TEST_DINT := 100;
	TestSuite.Test(__POUNAME()).AssertEqual(TEST_DINT, RawBuffer[TEST_LL+0]);
END_IF
END_METHOD

// AppendRight returns FALSE when element size doesn't match buffer element size
METHOD ReturnsFalseOnWrongSize
IF TestSuite.Test(__POUNAME()).ExecuteTest() THEN
	// Arrange
	fbAnyBuffer.Clear();
	WrongSizeElement := 100;  // INT is 2 bytes, buffer expects DINT (4 bytes)

	// Act - Pass an INT to a DINT buffer
	Success := fbAnyBuffer.PushRight(element := WrongSizeElement);

	// Assert
	TestSuite.Test(__POUNAME()).AssertEqual(TEST_BOOL_FALSE, Success);
END_IF
END_METHOD

// AppendRight returns TRUE when append succeeds
METHOD ReturnsTrueOnSuccess
IF TestSuite.Test(__POUNAME()).ExecuteTest() THEN
	// Arrange
	fbAnyBuffer.Clear();
	AppendedElement := 42;

	// Act
	Success := fbAnyBuffer.PushRight(element := AppendedElement);

	// Assert
	TestSuite.Test(__POUNAME()).AssertEqual(TEST_BOOL_TRUE, Success);
END_IF
END_METHOD

END_PROGRAM

// ---- UnitTests/AnyBuffer/TEST_AnyBuffer_ReplaceAtIndex.TcPOU
PROGRAM TEST_AnyBuffer_ReplaceAtIndex
VAR
	// Loop counter
	i						: DINT;
END_VAR

ReplaceAtBeginning();
ReplaceInMiddle();
ReplaceAtEnd();
ReturnsTrueOnSuccess();
ReturnsFalseOnNegativeIndex();
ReturnsFalseOnIndexAtCapacity();
ReturnsFalseOnIndexAboveCapacity();
WrongElementSize();
BufferUnchangedExceptIndex();
MetadataUnchanged();
MultipleReplacements();
ReplaceAllCapacityPositions();
ReplaceWithDifferentValues();
ReplaceSameIndexMultipleTimes();
ReplaceEmptyPosition();
ReplaceWhenBufferEmpty();

// All other elements remain unchanged after replace
METHOD BufferUnchangedExceptIndex
IF TestSuite.Test(__POUNAME()).ExecuteTest() THEN
	// Arrange - [100, 200, 300, 400, 500]
	fbAnyBuffer.Clear();
	FOR i := 1 TO 5 DO
		testElement := i * 100;
		fbAnyBuffer.PushRight(element := testElement);
	END_FOR

	// Act - Replace middle element (index 2)
	testElement := DINT#999;
	Success := fbAnyBuffer.ReplaceAtIndex(index := TEST_LL+2, element := testElement);

	// Assert - Only index 2 should be changed
	TestSuite.Test(__POUNAME()).AssertEqual(TEST_BOOL_TRUE, Success);
	TEST_DINT := 100;
	TestSuite.Test(__POUNAME()).AssertEqual(TEST_DINT, RawBuffer[TEST_LL+0]);
	TEST_DINT := 200;
	TestSuite.Test(__POUNAME()).AssertEqual(TEST_DINT, RawBuffer[TEST_LL+1]);
	TEST_DINT := 999;
	TestSuite.Test(__POUNAME()).AssertEqual(TEST_DINT, RawBuffer[TEST_LL+2]);
	TEST_DINT := 400;
	TestSuite.Test(__POUNAME()).AssertEqual(TEST_DINT, RawBuffer[TEST_LL+3]);
	TEST_DINT := 500;
	TestSuite.Test(__POUNAME()).AssertEqual(TEST_DINT, RawBuffer[TEST_LL+4]);
END_IF
END_METHOD

// ElementCount and all metadata remain unchanged after replace
METHOD MetadataUnchanged
IF TestSuite.Test(__POUNAME()).ExecuteTest() THEN
	// Arrange
	fbAnyBuffer.Clear();
	FOR i := 1 TO TEST_UL-TEST_LL+1 DO
		testElement := i * 100;
		fbAnyBuffer.PushRight(element := testElement);
	END_FOR
	TEST_DINT := 5;
	TestSuite.Test(__POUNAME()).AssertEqual(TEST_DINT, fbAnyBuffer.Metadata.elementCount);
	// Verify capacity was updated by PushRight
	TEST_DINT := 0;
	TestSuite.Test(__POUNAME()).AssertEqual(TEST_DINT, fbAnyBuffer.Metadata.capacity);

	// Act - Replace several elements
	testElement := DINT#111;
	Success := fbAnyBuffer.ReplaceAtIndex(index := TEST_LL, element := testElement);
	TestSuite.Test(__POUNAME()).AssertEqual(TEST_BOOL_TRUE, Success);

	testElement := DINT#333;
	Success := fbAnyBuffer.ReplaceAtIndex(index := TEST_LL+2, element := testElement);
	TestSuite.Test(__POUNAME()).AssertEqual(TEST_BOOL_TRUE, Success);

	testElement := DINT#555;
	Success := fbAnyBuffer.ReplaceAtIndex(index := TEST_LL+4, element := testElement);
	TestSuite.Test(__POUNAME()).AssertEqual(TEST_BOOL_TRUE, Success);

	// Assert - All metadata should be unchanged
	TEST_DINT := 5;
	TestSuite.Test(__POUNAME()).AssertEqual(TEST_DINT, fbAnyBuffer.Metadata.elementCount);
	TEST_DINT := 0;
	TestSuite.Test(__POUNAME()).AssertEqual(TEST_DINT, fbAnyBuffer.Metadata.capacity);
END_IF
END_METHOD

// Sequential replacements at different indices work correctly
METHOD MultipleReplacements
IF TestSuite.Test(__POUNAME()).ExecuteTest() THEN
	// Arrange
	fbAnyBuffer.Clear();
	FOR i := 1 TO TEST_UL-TEST_LL+1 DO
		testElement := i * 100;
		fbAnyBuffer.PushRight(element := testElement);
	END_FOR

	// Act - Replace multiple positions
	testElement := DINT#111;
	Success := fbAnyBuffer.ReplaceAtIndex(index := TEST_LL, element := testElement);
	TestSuite.Test(__POUNAME()).AssertEqual(TEST_BOOL_TRUE, Success);

	testElement := DINT#222;
	Success := fbAnyBuffer.ReplaceAtIndex(index := TEST_LL+1, element := testElement);
	TestSuite.Test(__POUNAME()).AssertEqual(TEST_BOOL_TRUE, Success);

	testElement := DINT#555;
	Success := fbAnyBuffer.ReplaceAtIndex(index := TEST_LL+4, element := testElement);
	TestSuite.Test(__POUNAME()).AssertEqual(TEST_BOOL_TRUE, Success);

	// Assert - All replacements should be successful
	TEST_DINT := 111;
	TestSuite.Test(__POUNAME()).AssertEqual(TEST_DINT, RawBuffer[TEST_LL]);
	TEST_DINT := 222;
	TestSuite.Test(__POUNAME()).AssertEqual(TEST_DINT, RawBuffer[TEST_LL+1]);
	TEST_DINT := 300;
	TestSuite.Test(__POUNAME()).AssertEqual(TEST_DINT, RawBuffer[TEST_LL+2]);
	TEST_DINT := 400;
	TestSuite.Test(__POUNAME()).AssertEqual(TEST_DINT, RawBuffer[TEST_LL+3]);
	TEST_DINT := 555;
	TestSuite.Test(__POUNAME()).AssertEqual(TEST_DINT, RawBuffer[TEST_LL+4]);
END_IF
END_METHOD

// Can replace every capacity position (0 to capacity-1)
METHOD ReplaceAllCapacityPositions
IF TestSuite.Test(__POUNAME()).ExecuteTest() THEN
	// Arrange - Fill buffer completely
	fbAnyBuffer.Clear();
	FOR i := 1 TO TEST_UL-TEST_LL+1 DO
		testElement := i * 100;
		fbAnyBuffer.PushRight(element := testElement);
	END_FOR

	// Act - Replace all capacity positions (0 through capacity-1 = 0 through 4)
	FOR i := TEST_LL TO TEST_UL DO
		testElement := (i-TEST_LL + 1) * 1000;
		Success := fbAnyBuffer.ReplaceAtIndex(index := TO_DINT(i), element := testElement);
		TestSuite.Test(__POUNAME()).AssertEqual(TEST_BOOL_TRUE, Success);
	END_FOR

	// Assert - All positions should be replaced
	TEST_DINT := 1000;
	TestSuite.Test(__POUNAME()).AssertEqual(TEST_DINT, RawBuffer[TEST_LL]);
	TEST_DINT := 2000;
	TestSuite.Test(__POUNAME()).AssertEqual(TEST_DINT, RawBuffer[TEST_LL+1]);
	TEST_DINT := 3000;
	TestSuite.Test(__POUNAME()).AssertEqual(TEST_DINT, RawBuffer[TEST_LL+2]);
	TEST_DINT := 4000;
	TestSuite.Test(__POUNAME()).AssertEqual(TEST_DINT, RawBuffer[TEST_LL+3]);
	TEST_DINT := 5000;
	TestSuite.Test(__POUNAME()).AssertEqual(TEST_DINT, RawBuffer[TEST_LL+4]);
	// Metadata unchanged
	TEST_DINT := 5;
	TestSuite.Test(__POUNAME()).AssertEqual(TEST_DINT, fbAnyBuffer.Metadata.elementCount);
END_IF
END_METHOD

// Replacing at index 0 updates first element correctly
METHOD ReplaceAtBeginning
IF TestSuite.Test(__POUNAME()).ExecuteTest() THEN
	// Arrange
	fbAnyBuffer.Clear();
	testElement := DINT#100;
	fbAnyBuffer.PushRight(element := testElement);
	testElement := DINT#200;
	fbAnyBuffer.PushRight(element := testElement);
	testElement := DINT#300;
	fbAnyBuffer.PushRight(element := testElement);

	// Act - Replace first element
	testElement := DINT#999;
	Success := fbAnyBuffer.ReplaceAtIndex(index := TEST_LL, element := testElement);

	// Assert
	TestSuite.Test(__POUNAME()).AssertEqual(TEST_BOOL_TRUE, Success);
	TEST_DINT := 999;
	TestSuite.Test(__POUNAME()).AssertEqual(TEST_DINT, RawBuffer[TEST_LL]);
	TEST_DINT := 200;
	TestSuite.Test(__POUNAME()).AssertEqual(TEST_DINT, RawBuffer[TEST_LL+1]);
	TEST_DINT := 300;
	TestSuite.Test(__POUNAME()).AssertEqual(TEST_DINT, RawBuffer[TEST_LL+2]);
	TEST_DINT := 3;
	TestSuite.Test(__POUNAME()).AssertEqual(TEST_DINT, fbAnyBuffer.Metadata.elementCount);
END_IF
END_METHOD

// Replacing at last capacity index updates last element
METHOD ReplaceAtEnd
IF TestSuite.Test(__POUNAME()).ExecuteTest() THEN
	// Arrange - fill buffer to capacity
	fbAnyBuffer.Clear();
	testElement := DINT#100;
	fbAnyBuffer.PushRight(element := testElement);
	testElement := DINT#200;
	fbAnyBuffer.PushRight(element := testElement);
	testElement := DINT#300;
	fbAnyBuffer.PushRight(element := testElement);
	testElement := DINT#400;
	fbAnyBuffer.PushRight(element := testElement);
	testElement := DINT#500;
	fbAnyBuffer.PushRight(element := testElement);

	// Act - Replace last capacity position (index 4 = capacity-1)
	testElement := DINT#999;
	Success := fbAnyBuffer.ReplaceAtIndex(index := TEST_LL+4, element := testElement);

	// Assert
	TestSuite.Test(__POUNAME()).AssertEqual(TEST_BOOL_TRUE, Success);
	TEST_DINT := 100;
	TestSuite.Test(__POUNAME()).AssertEqual(TEST_DINT, RawBuffer[TEST_LL]);
	TEST_DINT := 200;
	TestSuite.Test(__POUNAME()).AssertEqual(TEST_DINT, RawBuffer[TEST_LL+1]);
	TEST_DINT := 300;
	TestSuite.Test(__POUNAME()).AssertEqual(TEST_DINT, RawBuffer[TEST_LL+2]);
	TEST_DINT := 400;
	TestSuite.Test(__POUNAME()).AssertEqual(TEST_DINT, RawBuffer[TEST_LL+3]);
	TEST_DINT := 999;
	TestSuite.Test(__POUNAME()).AssertEqual(TEST_DINT, RawBuffer[TEST_LL+4]);
	// Metadata unchanged
	TEST_DINT := 5;
	TestSuite.Test(__POUNAME()).AssertEqual(TEST_DINT, fbAnyBuffer.Metadata.elementCount);
END_IF
END_METHOD

// Can replace position that was never filled (elementCount < index < capacity)
METHOD ReplaceEmptyPosition
IF TestSuite.Test(__POUNAME()).ExecuteTest() THEN
	// Arrange - only fill first 2 positions
	fbAnyBuffer.Clear();
	testElement := DINT#100;
	fbAnyBuffer.PushRight(element := testElement);
	testElement := DINT#200;
	fbAnyBuffer.PushRight(element := testElement);
	// elementCount = 2, but capacity = 5, so indices 2, 3, 4 are "empty"

	// Act - Replace position 3 (which was never logically filled)
	testElement := DINT#999;
	Success := fbAnyBuffer.ReplaceAtIndex(index := TEST_LL+3, element := testElement);

	// Assert - Should succeed because index 3 is within capacity
	TestSuite.Test(__POUNAME()).AssertEqual(TEST_BOOL_TRUE, Success);
	TEST_DINT := 999;
	TestSuite.Test(__POUNAME()).AssertEqual(TEST_DINT, RawBuffer[TEST_LL+3]);

	// Metadata should remain unchanged
	TEST_DINT := 2;
	TestSuite.Test(__POUNAME()).AssertEqual(TEST_DINT, fbAnyBuffer.Metadata.elementCount);
END_IF
END_METHOD

// Replacing at middle index updates correct element
METHOD ReplaceInMiddle
IF TestSuite.Test(__POUNAME()).ExecuteTest() THEN
	// Arrange
	fbAnyBuffer.Clear();
	testElement := DINT#100;
	fbAnyBuffer.PushRight(element := testElement);
	testElement := DINT#200;
	fbAnyBuffer.PushRight(element := testElement);
	testElement := DINT#300;
	fbAnyBuffer.PushRight(element := testElement);
	testElement := DINT#400;
	fbAnyBuffer.PushRight(element := testElement);

	// Act - Replace middle element (index 1)
	testElement := DINT#999;
	Success := fbAnyBuffer.ReplaceAtIndex(index := TEST_LL+1, element := testElement);

	// Assert
	TestSuite.Test(__POUNAME()).AssertEqual(TEST_BOOL_TRUE, Success);
	TEST_DINT := 100;
	TestSuite.Test(__POUNAME()).AssertEqual(TEST_DINT, RawBuffer[TEST_LL+0]);
	TEST_DINT := 999;
	TestSuite.Test(__POUNAME()).AssertEqual(TEST_DINT, RawBuffer[TEST_LL+1]);
	TEST_DINT := 300;
	TestSuite.Test(__POUNAME()).AssertEqual(TEST_DINT, RawBuffer[TEST_LL+2]);
	TEST_DINT := 400;
	TestSuite.Test(__POUNAME()).AssertEqual(TEST_DINT, RawBuffer[TEST_LL+3]);
	TEST_DINT := 4;
	TestSuite.Test(__POUNAME()).AssertEqual(TEST_DINT, fbAnyBuffer.Metadata.elementCount);
END_IF
END_METHOD

// Can overwrite same position repeatedly
METHOD ReplaceSameIndexMultipleTimes
IF TestSuite.Test(__POUNAME()).ExecuteTest() THEN
	// Arrange
	fbAnyBuffer.Clear();
	testElement := DINT#100;
	fbAnyBuffer.PushRight(element := testElement);
	testElement := DINT#200;
	fbAnyBuffer.PushRight(element := testElement);
	testElement := DINT#300;
	fbAnyBuffer.PushRight(element := testElement);

	// Act - Replace same index multiple times
	testElement := DINT#111;
	Success := fbAnyBuffer.ReplaceAtIndex(index := TEST_LL+1, element := testElement);
	TestSuite.Test(__POUNAME()).AssertEqual(TEST_BOOL_TRUE, Success);
	TEST_DINT := 111;
	TestSuite.Test(__POUNAME()).AssertEqual(TEST_DINT, RawBuffer[TEST_LL+1]);

	testElement := DINT#222;
	Success := fbAnyBuffer.ReplaceAtIndex(index := TEST_LL+1, element := testElement);
	TestSuite.Test(__POUNAME()).AssertEqual(TEST_BOOL_TRUE, Success);
	TEST_DINT := 222;
	TestSuite.Test(__POUNAME()).AssertEqual(TEST_DINT, RawBuffer[TEST_LL+1]);

	testElement := DINT#333;
	Success := fbAnyBuffer.ReplaceAtIndex(index := TEST_LL+1, element := testElement);
	TestSuite.Test(__POUNAME()).AssertEqual(TEST_BOOL_TRUE, Success);
	TEST_DINT := 333;
	TestSuite.Test(__POUNAME()).AssertEqual(TEST_DINT, RawBuffer[TEST_LL+1]);

	// Assert - Other elements unchanged, count unchanged
	TEST_DINT := 100;
	TestSuite.Test(__POUNAME()).AssertEqual(TEST_DINT, RawBuffer[TEST_LL+0]);
	TEST_DINT := 300;
	TestSuite.Test(__POUNAME()).AssertEqual(TEST_DINT, RawBuffer[TEST_LL+2]);
	TEST_DINT := 3;
	TestSuite.Test(__POUNAME()).AssertEqual(TEST_DINT, fbAnyBuffer.Metadata.elementCount);
END_IF
END_METHOD

// Replace succeeds even when elementCount = 0 (if index < capacity)
METHOD ReplaceWhenBufferEmpty
IF TestSuite.Test(__POUNAME()).ExecuteTest() THEN
	// Arrange - empty buffer (elementCount = 0)
	fbAnyBuffer.Clear();
	// Buffer is empty, but capacity is 5, so indices 0-4 are valid

	// Act - Replace at various positions in empty buffer
	testElement := DINT#111;
	Success := fbAnyBuffer.ReplaceAtIndex(index := TEST_LL, element := testElement);
	TestSuite.Test(__POUNAME()).AssertEqual(TEST_BOOL_TRUE, Success);
	TEST_DINT := 111;
	TestSuite.Test(__POUNAME()).AssertEqual(TEST_DINT, RawBuffer[TEST_LL]);

	testElement := DINT#333;
	Success := fbAnyBuffer.ReplaceAtIndex(index := TEST_LL+2, element := testElement);
	TestSuite.Test(__POUNAME()).AssertEqual(TEST_BOOL_TRUE, Success);
	TEST_DINT := 333;
	TestSuite.Test(__POUNAME()).AssertEqual(TEST_DINT, RawBuffer[TEST_LL+2]);

	testElement := DINT#555;
	Success := fbAnyBuffer.ReplaceAtIndex(index := TEST_LL+4, element := testElement);
	TestSuite.Test(__POUNAME()).AssertEqual(TEST_BOOL_TRUE, Success);
	TEST_DINT := 555;
	TestSuite.Test(__POUNAME()).AssertEqual(TEST_DINT, RawBuffer[TEST_LL+4]);

	// Metadata should remain unchanged (still empty from logical perspective)
	TEST_DINT := 0;
	TestSuite.Test(__POUNAME()).AssertEqual(TEST_DINT, fbAnyBuffer.Metadata.elementCount);
END_IF
END_METHOD

// Replace works with various data values
METHOD ReplaceWithDifferentValues
IF TestSuite.Test(__POUNAME()).ExecuteTest() THEN
	// Arrange
	fbAnyBuffer.Clear();
	FOR i := TEST_LL-TEST_LL+1  TO TEST_UL-TEST_LL+1 DO
		testElement := i * 100;
		fbAnyBuffer.PushRight(element := testElement);
	END_FOR

	// Act - Replace with various values (zero, negative, large)
	testElement := DINT#0;
	Success := fbAnyBuffer.ReplaceAtIndex(index := TEST_LL+0, element := testElement);
	TestSuite.Test(__POUNAME()).AssertEqual(TEST_BOOL_TRUE, Success);

	testElement := DINT#-999;
	Success := fbAnyBuffer.ReplaceAtIndex(index := TEST_LL+2, element := testElement);
	TestSuite.Test(__POUNAME()).AssertEqual(TEST_BOOL_TRUE, Success);

	testElement := DINT#2147483647;  // Max DINT
	Success := fbAnyBuffer.ReplaceAtIndex(index := TEST_LL+4, element := testElement);
	TestSuite.Test(__POUNAME()).AssertEqual(TEST_BOOL_TRUE, Success);

	// Assert - All values replaced correctly
	TEST_DINT := 0;
	TestSuite.Test(__POUNAME()).AssertEqual(TEST_DINT, RawBuffer[TEST_LL+0]);
	TEST_DINT := 200;
	TestSuite.Test(__POUNAME()).AssertEqual(TEST_DINT, RawBuffer[TEST_LL+1]);
	TEST_DINT := -999;
	TestSuite.Test(__POUNAME()).AssertEqual(TEST_DINT, RawBuffer[TEST_LL+2]);
	TEST_DINT := 400;
	TestSuite.Test(__POUNAME()).AssertEqual(TEST_DINT, RawBuffer[TEST_LL+3]);
	TEST_DINT := 2147483647;
	TestSuite.Test(__POUNAME()).AssertEqual(TEST_DINT, RawBuffer[TEST_LL+4]);
END_IF
END_METHOD

// FALSE returned when index > capacity
METHOD ReturnsFalseOnIndexAboveCapacity
IF TestSuite.Test(__POUNAME()).ExecuteTest() THEN
	// Arrange - capacity is 5
	fbAnyBuffer.Clear();
	testElement := DINT#100;
	fbAnyBuffer.PushRight(element := testElement);
	testElement := DINT#200;
	fbAnyBuffer.PushRight(element := testElement);

	// Act & Assert - Try index much larger than capacity
	testElement := DINT#999;
	Success := fbAnyBuffer.ReplaceAtIndex(index := TEST_UL+100, element := testElement);
	TestSuite.Test(__POUNAME()).AssertEqual(TEST_BOOL_FALSE, Success);

	// Act & Assert - Try another large index
	Success := fbAnyBuffer.ReplaceAtIndex(index := TEST_UL+10, element := testElement);
	TestSuite.Test(__POUNAME()).AssertEqual(TEST_BOOL_FALSE, Success);
END_IF
END_METHOD

// FALSE returned when index == capacity
METHOD ReturnsFalseOnIndexAtCapacity
IF TestSuite.Test(__POUNAME()).ExecuteTest() THEN
	// Arrange - capacity is 5
	fbAnyBuffer.Clear();
	testElement := DINT#100;
	fbAnyBuffer.PushRight(element := testElement);

	// Act - Try to replace beyond last index
	testElement := DINT#999;
	Success := fbAnyBuffer.ReplaceAtIndex(index := TEST_LL+5, element := testElement);

	// Assert
	TestSuite.Test(__POUNAME()).AssertEqual(TEST_BOOL_FALSE, Success);
END_IF
END_METHOD

// FALSE returned for negative index
METHOD ReturnsFalseOnNegativeIndex
IF TestSuite.Test(__POUNAME()).ExecuteTest() THEN
	// Arrange
	fbAnyBuffer.Clear();
	testElement := DINT#100;
	fbAnyBuffer.PushRight(element := testElement);

	// Act
	testElement := DINT#999;
	Success := fbAnyBuffer.ReplaceAtIndex(index := TEST_LL-1, element := testElement);

	// Assert
	TestSuite.Test(__POUNAME()).AssertEqual(TEST_BOOL_FALSE, Success);
	TEST_DINT := 1;
	TestSuite.Test(__POUNAME()).AssertEqual(TEST_DINT, fbAnyBuffer.Metadata.elementCount);
	TEST_DINT := 100;
	TestSuite.Test(__POUNAME()).AssertEqual(TEST_DINT, RawBuffer[TEST_LL+0]);
END_IF
END_METHOD

// Method returns TRUE when replace succeeds
METHOD ReturnsTrueOnSuccess
IF TestSuite.Test(__POUNAME()).ExecuteTest() THEN
	// Arrange
	fbAnyBuffer.Clear();
	testElement := DINT#100;
	fbAnyBuffer.PushRight(element := testElement);
	testElement := DINT#200;
	fbAnyBuffer.PushRight(element := testElement);

	// Act
	testElement := DINT#999;
	Success := fbAnyBuffer.ReplaceAtIndex(index := TEST_LL, element := testElement);

	// Assert
	TestSuite.Test(__POUNAME()).AssertEqual(TEST_BOOL_TRUE, Success);
END_IF
END_METHOD

// FALSE returned when element size doesn't match
METHOD WrongElementSize
IF TestSuite.Test(__POUNAME()).ExecuteTest() THEN
	// Arrange
	fbAnyBuffer.Clear();
	testElement := DINT#100;
	fbAnyBuffer.PushRight(element := testElement);

	// Act - Try to replace with wrong element size
	Success := fbAnyBuffer.ReplaceAtIndex(index := TEST_LL, element := WrongSizeElement);

	// Assert - Should fail (IN and DINT are different size)
	TestSuite.Test(__POUNAME()).AssertEqual(TEST_BOOL_FALSE, Success);

	// Verify buffer element count unchanged
	TEST_DINT := 1;
	TestSuite.Test(__POUNAME()).AssertEqual(TEST_DINT, fbAnyBuffer.Metadata.elementCount);
END_IF
END_METHOD

END_PROGRAM

// ---- _Mockups/Modules/ModuleCollection_Mockup.TcPOU
FUNCTION_BLOCK ModuleCollection_Mockup EXTENDS ModuleCollection<ApplicationBaseParameter.MaxCountInCollections>
VAR
END_VAR

METHOD GetInterfaceById : I_Module
VAR_INPUT
	Id : UDINT;
END_VAR

VAR
	Module : I_Module;
END_VAR
//__QUERYINTERFACE(Modules.GetItemById(Id), Module);

//GetInterfaceById := Module;
END_METHOD

END_FUNCTION_BLOCK
